// TIA Portal V16 export
// export: Created 2021-08-10T09:04:59.9476176Z, ExportSetting WithDefaults, WithReadOnly, DisplayName Totally Integrated Automation Portal, DisplayVersion V16, DisplayName TIA Portal Version Control Interface, DisplayVersion V16, DisplayName TIA Portal Openness, DisplayVersion V16, DisplayName TIA Portal Teamcenter Gateway, DisplayVersion V16, DisplayName SINAMICS Startdrive Advanced, DisplayVersion V16, DisplayName SINAMICS Startdrive G130, G150, S120, S150, SINAMICS MV, S210, DisplayVersion V16, DisplayName SINAMICS Startdrive G110M, G120, G120C, G120D, G120P, DisplayVersion V16, DisplayName STEP 7 Professional, DisplayVersion V16, DisplayName STEP 7 Safety, DisplayVersion V16, DisplayName WinCC Unified SCADA Engineering System, DisplayVersion V16
DATA_BLOCK "Program Logic_DB"   // DB2
{ S7_Optimized_Access := 'TRUE' }
VERSION : 0.1
// stored: AutoNumber true, CodeModifiedDate 2020-02-26T12:50:20.2800962Z, CompileDate 2021-07-03T08:38:45.0845051Z, CreationDate 2020-02-26T12:50:20.1014064Z, DBAccessibleFromOPCUA true, DownloadWithoutReinit false, InstanceOfName Program Logic, InstanceOfNumber 5, InstanceOfType FB, InterfaceModifiedDate 2020-02-26T11:20:20.4837101Z, IsConsistent true, IsKnowHowProtected false, IsRetainMemResEnabled false, MemoryReserve 100, ModifiedDate 2020-02-26T12:50:20.2800962Z, ParameterModified 2020-02-26T07:17:15.9384502Z, StructureModified 2020-02-26T11:20:20.4837101Z, UDAEnableTagReadback false
"Program Logic"
   // VAR
   //    StepSeq : "fbStepSequencer";
   //    CurrentStep { S7_SetPoint := 'True'} : Int;
   //    NextStep : Int;
   //    StepDone : Bool;
   // END_VAR
BEGIN
END_DATA_BLOCK
